FUNCTION_BLOCK TcoCr800_v_1_x_x EXTENDS TcoIo.TcoPnIoComponent  IMPLEMENTS TcoAbstractions.ITcoRobotics
VAR_INPUT
    inEnable : BOOL;
END_VAR
VAR_OUTPUT
END_VAR
VAR_IN_OUT
    inoData : TcoCr800_IO_v_1_x_x;
END_VAR
VAR
    

	{attribute addProperty Name "<#Status#>"}
    {attribute clr [ReadOnly()]}
    _status : TcoMitsubishiRobotics_Status_v_1_x_x;
	{attribute addProperty Name "<#Control#>"}
	_control 	: TcoMitsubishiRobotics_Control_v_1_x_x;
	{attribute addProperty Name "<#Config#>"}
    _config : TcoMitsubishiRobotics_Config_v_1_x_x;
	{attribute addProperty Name "<#PN Error#>"}
    {attribute clr [ReadOnly()]}
    _pnError : BOOL;

	_someTaskIsActive: BOOL;

	_stopTasksAreActive: BOOL;
END_VAR
VAR
	{attribute addProperty Name "<#Start at Main#>"}
    _startAtMainTask : StartAtMainTask(THIS^);
	
	 {attribute addProperty Name "<#Start motors and program#>"}
    _startMotorsAndProgramTask : StartMotorsAndProgramTask(THIS^);
	
	 {attribute addProperty Name "<#Start program#>"}
    _startProgramTask : StartProgramTask(THIS^);
	
	{attribute addProperty Name "<#Start motors#>"}
    _startMotorsTask : StartMotorsTask(THIS^);
	
  	{attribute addProperty Name "<#Start movements#>"}
    _startMovementsTask : StartMovementsTask(THIS^);
	
	{attribute addProperty Name "<#Start motors program and movements#>"}
    _startMotorsProgramAndMovementsTask : StartMotorsProgramAndMovementsTask(THIS^);
	
  	
	
	
	 {attribute addProperty Name "<#Stop movements#>"}
    _stopMovementsTask : StopMovementsTask(THIS^);

	 {attribute addProperty Name "<#Stop movenents and program#>"}
    _stopMovementsAndProgramTask : StopMovementsAndProgramTask(THIS^);
	
	{attribute addProperty Name "<#Stop program#>"}
    _stopProgramTask : StopMovementsAndProgramTask(THIS^);
	
	{attribute addProperty Name "<#Stop motors#>"}
    _stopMotorsTask : StopMotorsTask(THIS^);
	

    {attribute addProperty Name "<#Restore#>"}
    _restoreTask : TcoCore.TcoTask(THIS^);
	

  
   

  

END_VAR

VAR
	{attribute 'hide'}
	_sb : TcoCore.StringBuilder;
END_VAR

IF NOT __ISVALIDREF(inoData) THEN
    Messenger.Post('Invalid reference', TcoCore.eMessageCategory.ProgrammingError);
    RETURN;
END_IF

SUPER^(inPnIoBoxState := THIS^.inoData.PnIoBoxState,inPnIoBoxDiag := THIS^.inoData.PnIoBoxDiag);
_pnError:= not _profinetReady;


UpdateStatus();
_stopTasksAreActive :=  _stopMovementsTask.Busy 
			AND _stopMovementsAndProgramTask.Busy 
			AND _stopProgramTask.Busy
			AND _stopMotorsTask.Busy;
			
_startAtMainTask.Enabled:=NOT _stopTasksAreActive;
_startAtMainTask(inoConfig:=_config,inoControl:=_control,inoStatus:=_status);


_startProgramTask.Enabled:=NOT _stopTasksAreActive;
_startProgramTask(inoConfig:=_config,inoControl:=_control,inoStatus:=_status);

_startMotorsTask.Enabled:=NOT _stopTasksAreActive AND NOT _startMotorsProgramAndMovementsTask.Busy AND NOT _startMotorsAndProgramTask.Busy;
_startMotorsTask(inoConfig:=_config,inoControl:=_control,inoStatus:=_status);

_startMotorsAndProgramTask.Enabled:=NOT _stopTasksAreActive AND NOT _startProgramTask.Busy AND NOT _startMotorsTask.Busy;
_startMotorsAndProgramTask(inoConfig:=_config,inoControl:=_control,inoStatus:=_status);

_startMovementsTask.Enabled:=NOT _startMotorsProgramAndMovementsTask.Busy AND NOT _stopMotorsTask.Busy;
_startMovementsTask(inoConfig:=_config,inoControl:=_control,inoStatus:=_status);

_startMotorsProgramAndMovementsTask.Enabled:=NOT _startMovementsTask.Busy  AND NOT _stopMotorsTask.Busy;
_startMotorsProgramAndMovementsTask(refStartMotorsAndProgramTask:=_startMotorsAndProgramTask, inoConfig:=_config,inoControl:=_control,inoStatus:=_status);


_stopMovementsTask.Enabled:=TRUE;
_stopMovementsTask(inoConfig:=_config,inoControl:=_control,inoStatus:=_status);

_stopMotorsTask.Enabled:=TRUE;
_stopMotorsTask(inoConfig:=_config,inoControl:=_control,inoStatus:=_status);

_stopProgramTask.Enabled:=TRUE;
_stopProgramTask(inoConfig:=_config,inoControl:=_control,inoStatus:=_status);

_stopMovementsAndProgramTask.Enabled:=NOT _stopProgramTask.Busy AND NOT _stopProgramTask.Busy;
_stopMovementsAndProgramTask(inoConfig:=_config,inoControl:=_control,inoStatus:=_status);



//*************RESTORE********************

_restoreTask.Enabled := TRUE;
IF _restoreTask.Execute() THEN
	Restore();
	_restoreTask.DoneWhen(TRUE);
END_IF
//****************************************

_someTaskIsActive := _startAtMainTask.Busy 
					OR _startMotorsAndProgramTask.Busy
					OR _startMovementsTask.Busy
					OR _startMovementsTask.Busy
					OR _stopMovementsTask.Busy
					OR _stopMovementsAndProgramTask.Busy
					OR _stopProgramTask.Busy;
					

//do not publish diagnostic message when component is not used
IF _someTaskIsActive THEN

	IF(_status.State.EmgStop) THEN
		Messenger.Error('<#Emergency stop active#>');
	END_IF;
	IF(NOT _status.State.SafetyOk) THEN
		Messenger.Warning('<#Safety Error #>');
	END_IF;
	IF(_status.State.ProgExecError) THEN
		Messenger.Error('<#Program execution error see robot panel for details#>');
	END_IF;
  
END_IF;

IF(_status.State.Error) THEN Messenger.Error(_sb.Clear().Append('<#Drive error no #>').Append(UDINT_TO_STRING(_status.State.EventId)).Append(' |[[0]AdvancedDiagnosticMessage]|').Append('.').Append('For details see the service mode').ToString()); END_IF;


UpdateControl();

(*~
	<docu>
		<summary>
			Gets the configuration of the IRC 5. 					
		</summary>			
	</docu>	
~*)
PROPERTY Config : REFERENCE TO TcoMitsubishiRobotics_Config_v_1_x_x
GET
Config REF= _config;
END_GET
END_PROPERTY

METHOD FB_init : BOOL
VAR_INPUT
	bInitRetains : BOOL; // if TRUE, the retain variables are initialized (warm start / cold start)
	bInCopyCode : BOOL;  // if TRUE, the instance afterwards gets moved into the copy code (online change)
  	ParentObject : ITcoObject;	
END_VAR
END_METHOD

(*~
	<docu>
		<summary>
			Restores this instance to the Ready state. Can be called explicitly or from within one of the restore mechanisms.	
		</summary>			
	</docu>	
~*)
METHOD Restore : ITcoRestorable
RestoreTasks();
_control.ActionNo:=255;
_control.GlobalSpeed:=0;
_control.Interupt:=FALSE;
_control.LoadAndStartProg:=FALSE;
_control.LoadProg:=FALSE;
_control.MotorOff:=FALSE;
_control.MotorOn:=FALSE;
_control.MotorOnAndStart:=FALSE;
_control.PointNo:=0;
_control.QuickStop:=FALSE;
_control.ResetEmgStop:=FALSE;
_control.ResetError:=FALSE;
_control.SoftStop:=FALSE;
_control.StartAtMain:=FALSE;
_control.StartProgram:=FALSE;
_control.StopCycle:=FALSE;
_control.StopInstruction:=FALSE;
_control.StopProgram:=FALSE;
_control.LimitSpeed := FALSE;
_control.ToolNo:=0;
_control.WorkobjectNo:=0;
_control.PointNo:=0;
_control.UserSpecSpeed1:=0;
_control.UserSpecSpeed2:=0;
_control.Coordinates.X:=0;
_control.Coordinates.Y:=0;
_control.Coordinates.Z:=0;
_control.Coordinates.Rx:=0;
_control.Coordinates.Ry:=0;
_control.Coordinates.Rz:=0;
END_METHOD

METHOD INTERNAL RestoreTasks
//_resetTask.Restore();
_startAtMainTask.Restore();
_startMovementsTask.Restore();
_startProgramTask.Restore();
_startMotorsTask.Restore();
_stopMotorsTask.Restore();
_startMotorsProgramAndMovementsTask.Restore();
_stopMovementsTask.Restore();
_startMotorsAndProgramTask.Restore();
_stopMovementsAndProgramTask.Restore();
_stopProgramTask.Restore();
END_METHOD

(*~
	<docu>
		<summary>
		    Custom service (manual, maintenance) logic.
			This method must be implemented in derived class.
		</summary>			
	</docu>	
~*)
METHOD PROTECTED ServiceMode
END_METHOD

METHOD PUBLIC StartAtMain : TcoCore.ITcoTaskStatus
VAR_INPUT
END_VAR
StartAtMain:=_startAtMainTask.Invoke();
END_METHOD

PROPERTY StartAtMainTask : TcoCore.ITcoTaskStatus
GET
StartAtMainTask := _startAtMainTask;
END_GET
END_PROPERTY

METHOD PUBLIC StartMotors : TcoCore.ITcoTaskStatus
StartMotors:=_startMotorsTask.Invoke();
END_METHOD

METHOD StartMotorsAndProgram : TcoCore.ITcoTaskStatus
VAR_INPUT
END_VAR
StartMotorsAndProgram := THIS^._startMotorsAndProgramTask.Invoke();
END_METHOD

PROPERTY StartMotorsAndProgramTask : TcoCore.ITcoTaskStatus
GET
StartMotorsAndProgramTask := _startMotorsAndProgramTask;
END_GET
END_PROPERTY

METHOD PUBLIC StartMotorsProgramAndMovements : TcoCore.ITcoTaskStatus
VAR_INPUT
	inData : TcoRoboticsMovementsParams;
END_VAR
StartMotorsProgramAndMovements:=_startMotorsProgramAndMovementsTask.InvokeWithParams(inData);
END_METHOD

PROPERTY StartMotorsProgramAndMovementsTask : TcoCore.ITcoTaskStatus
GET
StartMotorsProgramAndMovementsTask := _startMotorsProgramAndMovementsTask;
END_GET
END_PROPERTY

PROPERTY StartMotorsTask : TcoCore.ITcoTaskStatus
GET
StartMotorsTask := _startMotorsTask;
END_GET
END_PROPERTY

METHOD PUBLIC StartMovements : TcoCore.ITcoTaskStatus
VAR_INPUT
	inData : TcoRoboticsMovementsParams;
END_VAR
StartMovements:=_startMovementsTask.InvokeWithParams(inData);
END_METHOD

PROPERTY StartMovementsTask : TcoCore.ITcoTaskStatus
GET
StartMovementsTask := _startMovementsTask;
END_GET
END_PROPERTY

METHOD PUBLIC StartProgram : TcoCore.ITcoTaskStatus
StartProgram:=_startProgramTask.Invoke();
END_METHOD

PROPERTY StartProgramTask : TcoCore.ITcoTaskStatus
GET
StartProgramTask := _startProgramTask;
END_GET
END_PROPERTY

(*~
	<docu>
		<summary>
			Gets the status of the IRC5. 					
		</summary>			
	</docu>	
~*)
PROPERTY Status : REFERENCE TO TcoMitsubishiRobotics_Status_v_1_x_x
GET
Status REF= _status;
END_GET
END_PROPERTY

METHOD PUBLIC StopMotors : TcoCore.ITcoTaskStatus
StopMotors:=_stopMotorsTask.Invoke();
END_METHOD

PROPERTY StopMotorsTask : TcoCore.ITcoTaskStatus
GET
StopMotorsTask := _stopMotorsTask;
END_GET
END_PROPERTY

METHOD PUBLIC StopMovements : TcoCore.ITcoTaskStatus
VAR_INPUT
	inStopType : eTcoRoboticsStopType;
END_VAR
StopMovements:=_stopMovementsTask.InvokeWithParams(inStopType);
END_METHOD

METHOD PUBLIC StopMovementsAndProgram : TcoCore.ITcoTaskStatus
VAR_INPUT
	inStopType : eTcoRoboticsStopType;
END_VAR
StopMovementsAndProgram:=_stopMovementsAndProgramTask.InvokeWithParams(inStopType);
END_METHOD

PROPERTY StopMovementsAndProgramTask : TcoCore.ITcoTaskStatus
GET
StopMovementsAndProgramTask := _stopMovementsAndProgramTask;
END_GET
END_PROPERTY

PROPERTY StopMovementsTask : TcoCore.ITcoTaskStatus
GET
StopMovementsTask := _stopMovementsTask;
END_GET
END_PROPERTY

METHOD PUBLIC StopProgram : TcoCore.ITcoTaskStatus
StopProgram:=_stopProgramTask.Invoke();
END_METHOD

PROPERTY StopProgramTask : TcoCore.ITcoTaskStatus
GET
StopProgramTask := _stopProgramTask;
END_GET
END_PROPERTY

METHOD INTERNAL UpdateControl
VAR_INPUT
END_VAR

VAR
	index: INT;
END_VAR
//SYSTEM OUTPUTS
index:=0;
inoData.Out.Outputs[index].0	:=		_control.Interupt;    
inoData.Out.Outputs[index].1	:=		_control.LoadProg;    
inoData.Out.Outputs[index].2 	:= 		_control.LoadAndStartProg; 
inoData.Out.Outputs[index].3 	:= 		_control.MotorOff;
inoData.Out.Outputs[index].4 	:= 		_control.MotorOn;   
inoData.Out.Outputs[index].5 	:= 		_control.MotorOnAndStart; 
inoData.Out.Outputs[index].6 	:= 		_control.ResetEmgStop;    
inoData.Out.Outputs[index].7 	:= 		_control.ResetError; 

index:=1;
inoData.Out.Outputs[index].0 	:= 		_control.StartProgram;    
inoData.Out.Outputs[index].1 	:= 		_control.StartAtMain;    
inoData.Out.Outputs[index].2 	:= 		_control.StopProgram;    
inoData.Out.Outputs[index].3 	:= 		_control.QuickStop;    
inoData.Out.Outputs[index].4 	:= 		_control.SoftStop;    
inoData.Out.Outputs[index].5 	:= 		_control.StopCycle;    
inoData.Out.Outputs[index].6 	:= 		_control.StopInstruction;    
inoData.Out.Outputs[index].7 	:= 		_control.LimitSpeed;    


	
//Tool signals
index:=2;
inoData.Out.Outputs[index].0 	:= 		_control.Tool_1_Retract;    
inoData.Out.Outputs[index].1 	:= 		_control.Tool_1_Extend;    
inoData.Out.Outputs[index].2	:= 		_control.Tool_2_Retract;    
inoData.Out.Outputs[index].3	:= 		_control.Tool_2_Extend;    
inoData.Out.Outputs[index].4	:= 		_control.Tool_3_Retract;    
inoData.Out.Outputs[index].5	:= 		_control.Tool_3_Extend;    
inoData.Out.Outputs[index].6 	:= 		_control.Tool_4_Retract;    
inoData.Out.Outputs[index].7	:= 		_control.Tool_4_Extend;    
//master mode  such as manual/auto ....
index:=3;
inoData.Out.Outputs[index]:= _control.MasterMode;
//zone
index:=5;
inoData.Out.Outputs[index]:= _control.Zone;
//position
index:=6;
inoData.Out.Outputs[index]:= _control.InPosition;

//
//Movement parameters
index:=7;
inoData.Out.Outputs[index]:= _control.ActionNo;
index:=8;
inoData.Out.Outputs[index]:= _control.GlobalSpeed;
index:=9;
inoData.Out.Outputs[index]:= _control.ToolNo;
index:=10;
inoData.Out.Outputs[index]:= _control.WorkobjectNo;
index:=11;
inoData.Out.Outputs[index]:= _control.PointNo;
index:=12;
TcoUtilities.TcoDintToBytes(inFormat:=TcoUtilities.eTcoDataFormat.LittleEndian,
							inValue:=REAL_TO_DINT(_control.UserSpecSpeed1),
							outByte0:=inoData.Out.Outputs[index],
							outByte1:=inoData.Out.Outputs[index+1],
							outByte2:=inoData.Out.Outputs[index+2],
							outByte3:=inoData.Out.Outputs[index+3]);
index:=16;
TcoUtilities.TcoDintToBytes(inFormat:=TcoUtilities.eTcoDataFormat.LittleEndian,
							inValue:=REAL_TO_DINT(_control.UserSpecSpeed2),
							outByte0:=inoData.Out.Outputs[index],
							outByte1:=inoData.Out.Outputs[index+1],
							outByte2:=inoData.Out.Outputs[index+2],
							outByte3:=inoData.Out.Outputs[index+3]);

////Coordinates
index:=20;
TcoUtilities.TcoDintToBytes(inFormat:=TcoUtilities.eTcoDataFormat.LittleEndian,
							inValue:=REAL_TO_DINT((_control.Coordinates.X+10000.0)*10000.0),
							outByte0:=inoData.Out.Outputs[index],
							outByte1:=inoData.Out.Outputs[index+1],
							outByte2:=inoData.Out.Outputs[index+2],
							outByte3:=inoData.Out.Outputs[index+3]);
index:=24;
TcoUtilities.TcoDintToBytes(inFormat:=TcoUtilities.eTcoDataFormat.LittleEndian,
							inValue:=REAL_TO_DINT((_control.Coordinates.Y+10000.0)*10000.0),
							outByte0:=inoData.Out.Outputs[index],
							outByte1:=inoData.Out.Outputs[index+1],
							outByte2:=inoData.Out.Outputs[index+2],
							outByte3:=inoData.Out.Outputs[index+3]);
index:=28;
TcoUtilities.TcoDintToBytes(inFormat:=TcoUtilities.eTcoDataFormat.LittleEndian,
							inValue:=REAL_TO_DINT((_control.Coordinates.Z+10000.0)*10000.0),
							outByte0:=inoData.Out.Outputs[index],
							outByte1:=inoData.Out.Outputs[index+1],
							outByte2:=inoData.Out.Outputs[index+2],
							outByte3:=inoData.Out.Outputs[index+3]);
index:=32;
TcoUtilities.TcoDintToBytes(inFormat:=TcoUtilities.eTcoDataFormat.LittleEndian,
							inValue:=REAL_TO_DINT((_control.Coordinates.Rx+360.0)*10000.0),
							outByte0:=inoData.Out.Outputs[index],
							outByte1:=inoData.Out.Outputs[index+1],
							outByte2:=inoData.Out.Outputs[index+2],
							outByte3:=inoData.Out.Outputs[index+3]);
index:=36;
TcoUtilities.TcoDintToBytes(inFormat:=TcoUtilities.eTcoDataFormat.LittleEndian,
							inValue:=REAL_TO_DINT((_control.Coordinates.Ry+360.0)*10000.0),
							outByte0:=inoData.Out.Outputs[index],
							outByte1:=inoData.Out.Outputs[index+1],
							outByte2:=inoData.Out.Outputs[index+2],
							outByte3:=inoData.Out.Outputs[index+3]);
index:=40;
TcoUtilities.TcoDintToBytes(inFormat:=TcoUtilities.eTcoDataFormat.LittleEndian,
							inValue:=REAL_TO_DINT((_control.Coordinates.Rz+360.0)*10000.0),
							outByte0:=inoData.Out.Outputs[index],
							outByte1:=inoData.Out.Outputs[index+1],
							outByte2:=inoData.Out.Outputs[index+2],
							outByte3:=inoData.Out.Outputs[index+3]);
END_METHOD

METHOD INTERNAL UpdateStatus
VAR
    _message : STRING(125);

	tempOut: BYTE;
	index: INT;
	_bytes: DINT;
END_VAR
//SYSTEM INPUTS
index:=0;
_status.State.AutoOn := inoData.In.Inputs[index].0;
_status.State.CycleOn := inoData.In.Inputs[index].1;
_status.State.EmgStop := inoData.In.Inputs[index].2;
_status.State.Error := inoData.In.Inputs[index].3;
_status.State.MoveActive := inoData.In.Inputs[index].4;
_status.State.MoveInactive := inoData.In.Inputs[index].5;
_status.State.MotorOff := inoData.In.Inputs[index].6;
_status.State.MotorOn := inoData.In.Inputs[index].7;

index:=1;
_status.State.MotorOffState := inoData.In.Inputs[index].0;
_status.State.MotorOnState := inoData.In.Inputs[index].1;
_status.State.ProgExecError := inoData.In.Inputs[index].2;
_status.State.SafetyOk := inoData.In.Inputs[index].3;
_status.State.SystemInputBusy := inoData.In.Inputs[index].4;
_status.State.PpMoved := inoData.In.Inputs[index].5;
_status.State.MotionSupervision := inoData.In.Inputs[index].6;
_status.State.BatteryLow := inoData.In.Inputs[index].7;


//Area/positions flags this  should be obsolete because Zones and InPosition is used as byte below
index:=2;
_status.State.InArea_1 := inoData.In.Inputs[index].0;
_status.State.InArea_2 := inoData.In.Inputs[index].1;
_status.State.InArea_3 := inoData.In.Inputs[index].2;
_status.State.InArea_4 := inoData.In.Inputs[index].3;
_status.State.InPosition_1 := inoData.In.Inputs[index].4;
_status.State.InPosition_2 := inoData.In.Inputs[index].5;
_status.State.InPosition_3 := inoData.In.Inputs[index].6;
_status.State.InPosition_4 := inoData.In.Inputs[index].7;
//
//Tool signals
index:=3;
_status.State.Tool_1_Retract := inoData.In.Inputs[index].0;
_status.State.Tool_1_Extend := inoData.In.Inputs[index].1;
_status.State.Tool_2_Retract := inoData.In.Inputs[index].2;
_status.State.Tool_2_Extend := inoData.In.Inputs[index].3;
_status.State.Tool_3_Retract := inoData.In.Inputs[index].4;
_status.State.Tool_3_Extend := inoData.In.Inputs[index].5;
_status.State.Tool_4_Retract := inoData.In.Inputs[index].6;
_status.State.Tool_4_Extend := inoData.In.Inputs[index].7;

//Safety signals
index:=4;
_status.State.AutoStop_1 := inoData.In.Inputs[index].0;
_status.State.AutoStop_2 := inoData.In.Inputs[index].1;
_status.State.EmergencyStop_1 := inoData.In.Inputs[index].2;
_status.State.EmergencyStop_2 := inoData.In.Inputs[index].3;
_status.State.GeneralStop_1 := inoData.In.Inputs[index].4;
_status.State.GeneralStop_2 := inoData.In.Inputs[index].5;
_status.State.Enable_1 := inoData.In.Inputs[index].6;
_status.State.Enable_2 := inoData.In.Inputs[index].7;

index:=5;
_status.State.Zone:= inoData.In.Inputs[index];
index:=6;
_status.State.InPosition:= inoData.In.Inputs[index];

//Movement parameters
index:=7;
_status.State.ActionNo:= inoData.In.Inputs[index];
index:=8;
_status.State.GlobalSpeed:= inoData.In.Inputs[index];
index:=9;
_status.State.ToolNo:= inoData.In.Inputs[index];
index:=10;
_status.State.WorkobjectNo:= inoData.In.Inputs[index];
index:=11;
_status.State.PointNo:= inoData.In.Inputs[index];
index:=12;
_status.State.UserSpecSpeed1:=TcoUtilities.TcoBytesToDint (inFormat:=TcoUtilities.eTcoDataFormat.LittleEndian,
															inByte0:= inoData.In.Inputs[index],
															inByte1:= inoData.In.Inputs[index+1],
															inByte2:= inoData.In.Inputs[index+2],
															inByte3:= inoData.In.Inputs[index+3]);
index:=16;
_status.State.UserSpecSpeed2:=TcoUtilities.TcoBytesToDint (inFormat:=TcoUtilities.eTcoDataFormat.LittleEndian,
															inByte0:= inoData.In.Inputs[index],
															inByte1:= inoData.In.Inputs[index+1],
															inByte2:= inoData.In.Inputs[index+2],
															inByte3:= inoData.In.Inputs[index+3]);
															
index:=20;
_bytes:=TcoUtilities.TcoBytesToDint (inFormat:=TcoUtilities.eTcoDataFormat.LittleEndian,
															inByte0:= inoData.In.Inputs[index],
															inByte1:= inoData.In.Inputs[index+1],
															inByte2:= inoData.In.Inputs[index+2],
															inByte3:= inoData.In.Inputs[index+3]);

_status.State.Coordinates.X:=(DINT_TO_REAL(_bytes)/10000.0)-10000.0;

index:=24;
_bytes:=TcoUtilities.TcoBytesToDint (inFormat:=TcoUtilities.eTcoDataFormat.LittleEndian,
															inByte0:= inoData.In.Inputs[index],
															inByte1:= inoData.In.Inputs[index+1],
															inByte2:= inoData.In.Inputs[index+2],
															inByte3:= inoData.In.Inputs[index+3]);

_status.State.Coordinates.Y:=(DINT_TO_REAL(_bytes)/10000.0)-10000.0;

index:=28;
_bytes:=TcoUtilities.TcoBytesToDint (inFormat:=TcoUtilities.eTcoDataFormat.LittleEndian,
															inByte0:= inoData.In.Inputs[index],
															inByte1:= inoData.In.Inputs[index+1],
															inByte2:= inoData.In.Inputs[index+2],
															inByte3:= inoData.In.Inputs[index+3]);

_status.State.Coordinates.Z:=(DINT_TO_REAL(_bytes)/10000.0)-10000.0;

index:=32;															
_bytes:=TcoUtilities.TcoBytesToDint (inFormat:=TcoUtilities.eTcoDataFormat.LittleEndian,
															inByte0:= inoData.In.Inputs[index],
															inByte1:= inoData.In.Inputs[index+1],
															inByte2:= inoData.In.Inputs[index+2],
															inByte3:= inoData.In.Inputs[index+3]);

_status.State.Coordinates.Rx:=(DINT_TO_REAL(_bytes)/10000.0)-360.0;

index:=36;
_bytes:=TcoUtilities.TcoBytesToDint (inFormat:=TcoUtilities.eTcoDataFormat.LittleEndian,
															inByte0:= inoData.In.Inputs[index],
															inByte1:= inoData.In.Inputs[index+1],
															inByte2:= inoData.In.Inputs[index+2],
															inByte3:= inoData.In.Inputs[index+3]);

_status.State.Coordinates.Ry:=(DINT_TO_REAL(_bytes)/10000.0)-360.0;

index:=40;
_bytes:=TcoUtilities.TcoBytesToDint (inFormat:=TcoUtilities.eTcoDataFormat.LittleEndian,
															inByte0:= inoData.In.Inputs[index],
															inByte1:= inoData.In.Inputs[index+1],
															inByte2:= inoData.In.Inputs[index+2],
															inByte3:= inoData.In.Inputs[index+3]);

_status.State.Coordinates.Rz:=(DINT_TO_REAL(_bytes)/10000.0)-360.0;

index:=44;
_status.State.EventId:=TcoUtilities.TcoBytesToUDint (inFormat:=TcoUtilities.eTcoDataFormat.LittleEndian,
															inByte0:= inoData.In.Inputs[index],
															inByte1:= inoData.In.Inputs[index+1],
															inByte2:= inoData.In.Inputs[index+2],
															inByte3:= inoData.In.Inputs[index+3]);
END_METHOD

END_FUNCTION_BLOCK

(* stored: Version 1.1.0.1, ProductVersion 3.1.4024.12
   POU TcoCr800_v_1_x_x: Id {74b4ebc3-5b27-0a8f-2e6a-4eb1c4b210b2}, SpecialFunc None
   Folder Operations: Id {29d0d0e7-a391-03ad-2cac-68a6277da04b}
   Folder Task: Id {7dfeed1c-cda6-0dca-00d3-352e4feb8268}
   Property Config: Id {1a7a2474-a36b-098e-3034-5392cd841022}
   Get Get: Id {c9812583-2a1f-007a-1a76-e3a4fb32a803}
   Method FB_init: Id {38bfdeba-6232-0954-0701-387a681e834f}
   Method Restore: Id {d363ee24-34c7-0d8f-194e-b44d3f60cfa7}
   Method RestoreTasks: Id {33cc2c1d-106d-09c5-2090-55d489e8f08d}
   Method ServiceMode: Id {0ef2c3dc-7ed6-0556-261f-e54f8f20f0ab}
   Method StartAtMain: Id {6e7d70ea-7506-068e-2b8e-913fa2071119}
   Property StartAtMainTask: Id {3572e1bb-4932-0f7d-1030-6cd884430a78}
   Get Get: Id {f0b8bec9-70a3-0eab-181d-44369cb0f54e}
   Method StartMotors: Id {04f132c9-580d-0da9-1368-00c9546eeda4}
   Method StartMotorsAndProgram: Id {4a958ada-3ba7-0eb3-18f7-8142a2d362d1}
   Property StartMotorsAndProgramTask: Id {17e1d713-832b-03e9-1388-26310c65ba24}
   Get Get: Id {981fdc8e-c2a7-0009-263a-a5cb8df68745}
   Method StartMotorsProgramAndMovements: Id {e4ad34ef-84fd-0acf-1a63-f92a4a17a70c}
   Property StartMotorsProgramAndMovementsTask: Id {9f131e0f-910d-0dce-03a3-710bfa153d9a}
   Get Get: Id {3cd8937f-9f3a-0784-1369-926264c4b363}
   Property StartMotorsTask: Id {449dcdea-162e-0f68-26f4-c1fcb74138e1}
   Get Get: Id {a7b3f1d6-00e9-05e1-03a7-33f2da04c751}
   Method StartMovements: Id {a49fd687-f06d-0526-2635-c12e6112370a}
   Property StartMovementsTask: Id {498938f1-6399-0f05-38f6-68a5c4709933}
   Get Get: Id {0618238a-0974-071b-03d0-7e1794aa937f}
   Method StartProgram: Id {9b5b1463-9e51-0403-1386-25a54b78e848}
   Property StartProgramTask: Id {89e36195-a370-0c02-00d3-0430a186e225}
   Get Get: Id {80e45f2d-2e4e-0b16-36b2-460adedebf62}
   Property Status: Id {2d567d93-caf0-029a-360b-e17d83304f54}
   Get Get: Id {d7ef5b46-ab1b-024c-392d-9338eec7b11d}
   Method StopMotors: Id {836faee1-39ce-0fc5-3111-f10b4ad8ac97}
   Property StopMotorsTask: Id {24085091-1e0c-0c02-231b-dacda648c233}
   Get Get: Id {d6116290-18fd-0e2f-02b9-1ec23fba134d}
   Method StopMovements: Id {c915c105-f8e2-0894-2582-8c35284b44aa}
   Method StopMovementsAndProgram: Id {0fe7b92f-5877-0f63-295f-93eb07bd9e57}
   Property StopMovementsAndProgramTask: Id {a7efe5a3-b705-0d1d-3a31-f32a146b9278}
   Get Get: Id {d4bc0e46-e9a5-0d72-0ecf-7ccacc68e1b7}
   Property StopMovementsTask: Id {f7fada54-778f-06d5-1771-3499a26bacfc}
   Get Get: Id {c26caaf6-6299-0285-0962-8b4683b246c9}
   Method StopProgram: Id {12269af9-210f-0447-2af4-4e82f9fba185}
   Property StopProgramTask: Id {d8e3a7a4-25de-0006-0b74-b877cb39cde9}
   Get Get: Id {e0ed5ba0-96fb-0aec-2b0e-c8c95b46bfc6}
   Method UpdateControl: Id {6fa96b3c-54eb-06ee-2229-f662501a121c}
   Method UpdateStatus: Id {f412110d-4f6b-05c1-3bc2-6714c71388b1} *)
